ABB RobotStudio station: Demo FlexLoader.rspag

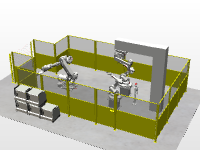
--- station ---
Station Demo FlexLoader (saved by RobotStudio 6.4.7096.126)
Controller Flexloader
  mechanical unit ROB_1: IRB6700_175_305__R1, 6 joints, base frame (0, 0, 0) mm
  mechanical unit ROB_2: IRB1600_6_145__R2, 6 joints, base frame (3100, -700, 540) mm, rotated rx 0 ry 0 rz 180 deg
  mechanical unit ROB_3: IRB1600_6_145__R3, 6 joints, base frame (3100, 700, 540) mm, rotated rx 0 ry 0 rz 180 deg
  mechanical unit ROB_4: IRB1600_6_145__R4, 6 joints, base frame (3100, 0, 2967) mm, rotated rx 180 ry 0 rz 180 deg
Layout (positions relative to the parent item):
  - PKI_500_di_M2001_R2 [mechanism, from Tools\PKI_500_di_M2001.rslib] at (2798.48, -669.1, 1835.93) mm, rotated rx 133.14 ry 80.29 rz -55.34 deg
  - PKI_500_di_M2001_R3 [mechanism, from Tools\PKI_500_di_M2001.rslib] at (2852.02, 663.13, 1854.7) mm, rotated rx -145.04 ry 81.85 rz 49.38 deg
  - PKI_500_di_M2001_R4 [mechanism, from Tools\PKI_500_di_M2001.rslib] at (3569.99, -25.32, 1662.65) mm, rotated rx 170.83 ry -31.84 rz -4.26 deg
  - balk [part] at (-1606.02, -38.05, 675.61) mm, rotated rx -179.44 ry -15.29 rz 176.39 deg
  - FixColumn [part] at (4831, 233, -8) mm, rotated rx 0 ry 0 rz -90 deg
  - RobotStand_2 [part] at (3123, -700, 0) mm, rotated rx 0 ry 0 rz 180 deg
  - RobotStand_3 [part] at (3130, 700, 0) mm, rotated rx 0 ry 0 rz 180 deg
  - IRC5_FlexController_1 [part, from Equipment\IRC5_Control-Module.rslib] at (0, -3200, 100) mm, rotated rx 90 ry 0 rz 0 deg
  - IRC5_DriveModule_1 [part, from Equipment\IRC5_Drive-Module.rslib] at (-750, -3200, 100) mm, rotated rx 90 ry 0 rz 0 deg
  - IRC5_DriveModule_2 [part, from Equipment\IRC5_Drive-Module.rslib] at (-750, -3200, 750) mm, rotated rx 90 ry 0 rz 0 deg
  - IRC5_DriveModule_3 [part, from Equipment\IRC5_Drive-Module.rslib] at (0, -3200, 750) mm, rotated rx 90 ry 0 rz 0 deg
  - IRC5_DriveModule_4 [part, from Equipment\IRC5_Drive-Module.rslib] at (750, -3200, 100) mm, rotated rx 90 ry 0 rz 0 deg
  - IRB1600_6_145__R2 [mechanism, from Robots\IRB1600_6_145_G_02.rslib] at (3100, -700, 540) mm, rotated rx 0 ry 0 rz 180 deg; joint values [-0.0917, -0.6874, 0.2096, -0.087, 0.5953, 0.202] (rad or m)
  - IRB1600_6_145__R3 [mechanism, from Robots\IRB1600_6_145_G_02.rslib] at (3100, 700, 540) mm, rotated rx 0 ry 0 rz 180 deg; joint values [0.1133, -0.7396, 0.1798, 0.2099, 0.6882, -0.2606] (rad or m)
  - IRB1600_6_145__R4 [mechanism, from Robots\IRB1600_6_145_G_02.rslib] at (3100, 0, 2967) mm, rotated rx 180 ry 0 rz 180 deg; joint values [0.0285, -1.3249, -0.0923, 0.2805, -0.7223, 2.9683] (rad or m)
  - IRB6700_175_305__R1 [mechanism, from Robots\IRB6700_175_305__04.rslib] at (0, 0, 0) mm; joint values [0.0254, -0.5043, -3.1116, -0.0184, -0.8299, 0.0976] (rad or m)
  - Fence [graphiccomponentgroup]
    - Segment 1 [part]
    - Segment 2 [part]
    - Segment 3 [part]
    - Segment 4 [part]
    - Segment 5 [part]
    - Segment 6 [part]
    - Segment 7 [part]
    - Segment 8 [part]
    - Segment 9 [part]
    - Segment 10 [part]
    - Segment 11 [part]
    - Segment 12 [part]
    - Segment 13 [part]
    - Segment 14 [part]
    - Segment 15 [part]
    - Segment 16 [part]
    - Segment 17 [part]
  - Floor [part]
  - TSC2013 [mechanism] at (3966.38, 33.42, 0) mm; joint values [1.225] (rad or m)
      links: L1, L2
  - LightGuard [graphiccomponentgroup]
    - GeneratedPart [part] at (-3200, -1000, 200) mm, rotated rx 0 ry 90 rz 90 deg
    - GeneratedPart [part] at (-3200, -1000, 250) mm, rotated rx 0 ry 90 rz 90 deg
    - GeneratedPart [part] at (-3200, -1000, 300) mm, rotated rx 0 ry 90 rz 90 deg
    - GeneratedPart [part] at (-3200, -1000, 350) mm, rotated rx 0 ry 90 rz 90 deg
    - GeneratedPart [part] at (-3200, -1000, 400) mm, rotated rx 0 ry 90 rz 90 deg
    - GeneratedPart [part] at (-3200, -1000, 450) mm, rotated rx 0 ry 90 rz 90 deg
    - GeneratedPart [part] at (-3200, -1000, 500) mm, rotated rx 0 ry 90 rz 90 deg
    - GeneratedPart [part] at (-3200, -1000, 550) mm, rotated rx 0 ry 90 rz 90 deg
    - GeneratedPart [part] at (-3200, -1000, 600) mm, rotated rx 0 ry 90 rz 90 deg
    - GeneratedPart [part] at (-3200, -1000, 650) mm, rotated rx 0 ry 90 rz 90 deg
    - GeneratedPart [part] at (-3200, -1000, 700) mm, rotated rx 0 ry 90 rz 90 deg
    - GeneratedPart [part] at (-3200, -1000, 750) mm, rotated rx 0 ry 90 rz 90 deg
    - GeneratedPart [part] at (-3200, -1000, 800) mm, rotated rx 0 ry 90 rz 90 deg
    - GeneratedPart [part] at (-3200, -1000, 850) mm, rotated rx 0 ry 90 rz 90 deg
    - GeneratedPart [part] at (-3200, -1000, 900) mm, rotated rx 0 ry 90 rz 90 deg
    - GeneratedPart [part] at (-3200, -1000, 950) mm, rotated rx 0 ry 90 rz 90 deg
    - GeneratedPart [part] at (-3200, -1000, 1000) mm, rotated rx 0 ry 90 rz 90 deg
    - GeneratedPart [part] at (-3200, -1000, 1050) mm, rotated rx 0 ry 90 rz 90 deg
    - GeneratedPart [part] at (-3200, -1000, 1100) mm, rotated rx 0 ry 90 rz 90 deg
    - GeneratedPart [part] at (-3200, -1000, 1150) mm, rotated rx 0 ry 90 rz 90 deg
    - GeneratedPart [part] at (-3200, -1000, 1200) mm, rotated rx 0 ry 90 rz 90 deg
    - GeneratedPart [part] at (-3200, -1000, 1250) mm, rotated rx 0 ry 90 rz 90 deg
    - GeneratedPart [part] at (-3200, -1000, 1300) mm, rotated rx 0 ry 90 rz 90 deg
    - GeneratedPart [part] at (-3200, -1000, 1350) mm, rotated rx 0 ry 90 rz 90 deg
    - GeneratedPart [part] at (-3200, -1000, 1400) mm, rotated rx 0 ry 90 rz 90 deg
    - GeneratedPart [part] at (-3200, -1000, 1450) mm, rotated rx 0 ry 90 rz 90 deg
    - GeneratedPart [part] at (-3200, -1000, 1500) mm, rotated rx 0 ry 90 rz 90 deg
    - GeneratedPart [part] at (-3200, -1000, 1550) mm, rotated rx 0 ry 90 rz 90 deg
    - GeneratedPart [part] at (-3200, -1000, 1600) mm, rotated rx 0 ry 90 rz 90 deg
    - GeneratedPart [part] at (-3200, -1000, 1650) mm, rotated rx 0 ry 90 rz 90 deg
    - GeneratedPart [part] at (-3200, -1000, 1700) mm, rotated rx 0 ry 90 rz 90 deg
    - GeneratedPart [part] at (-3200, -1000, 1750) mm, rotated rx 0 ry 90 rz 90 deg
    - light_guard1 [part] at (-3200, -1000, 0) mm, rotated rx 0 ry 0 rz 90 deg
    - light_guard2 [part] at (-3200, 1000, 0) mm, rotated rx 0 ry 0 rz 90 deg
  - R1 [frame] at (3100, -700, 540) mm, rotated rx 0 ry 0 rz 180 deg
  - R2 [frame] at (3100, 700, 540) mm, rotated rx 0 ry 0 rz 180 deg
  - R3 [frame] at (3100, 0, 2967) mm, rotated rx 180 ry 0 rz 180 deg
  - R4 [frame]
  - Frame_5 [frame] at (1912, 0, 2055) mm, rotated rx 0 ry 90 rz 0 deg
  - Frame_1 [frame] at (-1606.02, -38.05, 675.61) mm, rotated rx -179.44 ry -15.29 rz 176.39 deg
  - Frame_2 [frame]
Attachment: PKI_500_di_M2001_R2 is attached to IRB1600_6_145__R2 / Link6
Attachment: PKI_500_di_M2001_R3 is attached to IRB1600_6_145__R3 / Link6
Attachment: PKI_500_di_M2001_R4 is attached to IRB1600_6_145__R4 / Link6
Attachment: balk is attached to IRB6700_175_305__R1 / Link6
Targets, tools, work objects and paths stored in the station and not in the controller backup, written as RAPID:
! task T_ROB1
MODULE Module1
  CONST robtarget Target_10:=[[1912,0,2055],[0.707106781,0,0.707106781,0],[0,0,0,0],[9E+09,9E+09,9E+09,9E+09,9E+09,9E+09]];
  VAR syncident ident1;
  VAR syncident ident2;
  VAR syncident ident3;
  VAR syncident ident4;
  VAR syncident ident5;
  VAR syncident ident6;
  VAR syncident ident7;
  VAR syncident ident8;
  VAR syncident ident9;
ENDMODULE

! task T_ROB2
MODULE Module1
  VAR syncident ident1;
  VAR syncident ident2;
  VAR syncident ident3;
  VAR syncident ident4;
  VAR syncident ident5;
  VAR syncident ident6;
  VAR syncident ident7;
  VAR syncident ident8;
  VAR syncident ident9;
  VAR syncident identUnder1;
  VAR syncident identUnder2;
  VAR syncident identEdge1;
  VAR syncident identEdge2;
  VAR syncident identCurve1;
  VAR syncident identCurve2;
  VAR syncident identBack1;
  VAR syncident identBack2;
  VAR syncident identTop1;
  VAR syncident identTop2;
  VAR syncident identRing1;
  VAR syncident identRing2;
ENDMODULE

! task T_ROB3
MODULE Module1
  VAR syncident ident1;
  VAR syncident ident2;
  VAR syncident ident3;
  VAR syncident ident4;
  VAR syncident ident5;
  VAR syncident ident6;
  VAR syncident ident7;
  VAR syncident ident8;
  VAR syncident ident9;
  VAR syncident identUnder1;
  VAR syncident identUnder2;
  VAR syncident identEdge1;
  VAR syncident identEdge2;
  VAR syncident identCurve1;
  VAR syncident identCurve2;
  VAR syncident identBack1;
  VAR syncident identBack2;
  VAR syncident identTop1;
  VAR syncident identTop2;
  VAR syncident identRing1;
  VAR syncident identRing2;
ENDMODULE

! task T_ROB4
MODULE module1
  VAR syncident ident1;
  VAR syncident ident2;
  VAR syncident ident3;
  VAR syncident ident4;
  VAR syncident ident5;
  VAR syncident ident6;
  VAR syncident ident7;
  VAR syncident ident8;
  VAR syncident ident9;
  VAR syncident identEdge1;
  VAR syncident identEdge2;
  VAR syncident identTop1;
  VAR syncident identTop2;
ENDMODULE


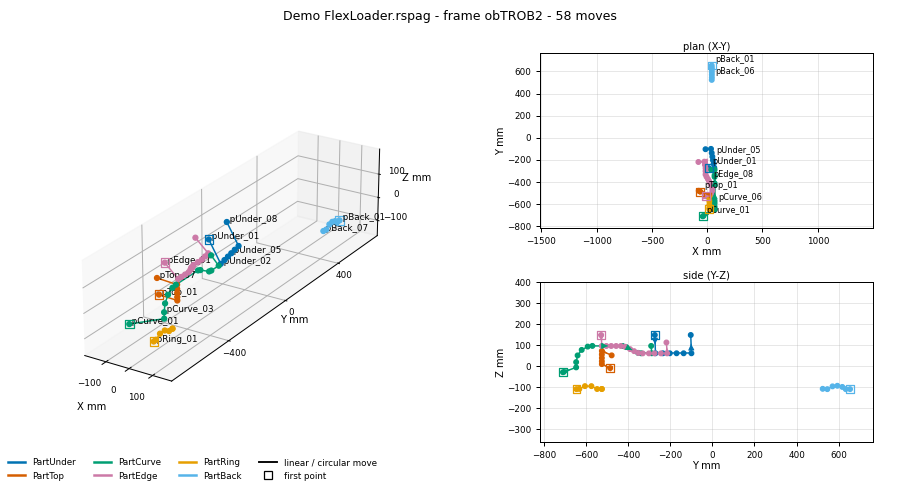
[picture p0: tool path of Demo FlexLoader.rspag in frame obTROB2, 58 of 166 moves have a stored position in this frame; points joined in program order, loops and branches not executed]
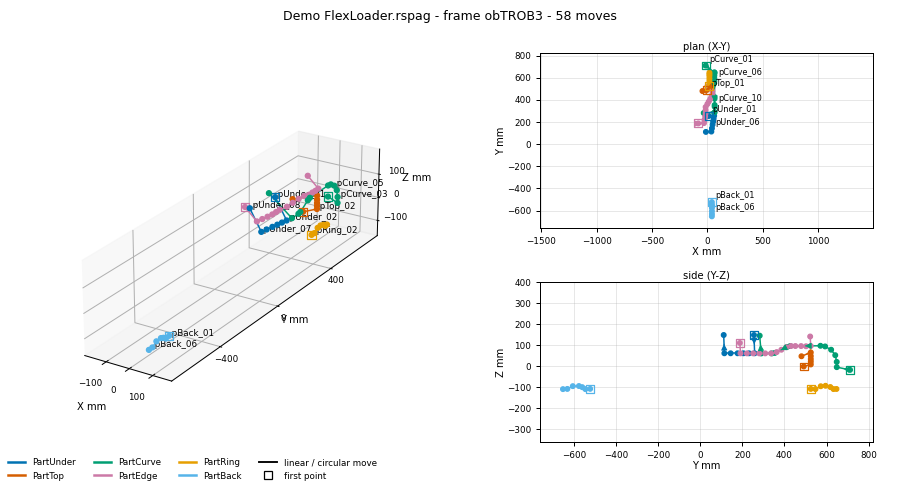
[picture p1: tool path of Demo FlexLoader.rspag in frame obTROB3, 58 of 166 moves have a stored position in this frame; points joined in program order, loops and branches not executed]
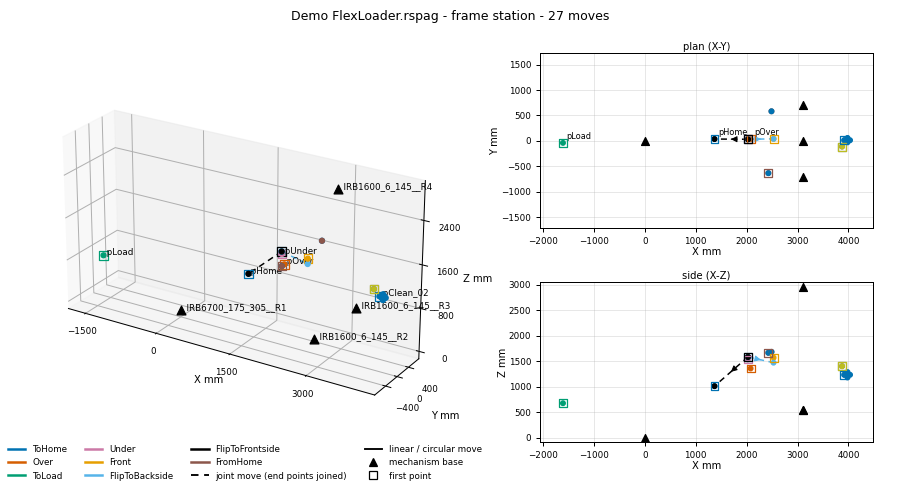
[picture p2: tool path of Demo FlexLoader.rspag in frame station, 27 of 166 moves have a stored position in this frame; points joined in program order, loops and branches not executed]
--- Backups/Flexloader/RAPID/TASK1/PROGMOD/Module1.mod ---
%%%
   VERSION: 1
   LANGUAGE: ENGLISH
%%%

MODULE Module1
	VAR syncident ident1;
	PERS tasks task1{4}:=[["T_ROB1"],["T_ROB2"],["T_ROB3"],["T_ROB4"]];
	VAR syncident ident2;
	VAR syncident ident3;
	VAR syncident ident4;
	VAR syncident ident5;
	VAR syncident ident6;
	PERS tasks task4{3}:=[["T_ROB1"],["T_ROB2"],["T_ROB3"]];
	VAR syncident ident7;
	VAR syncident ident8;
	VAR syncident ident9;
	CONST robtarget pHome:=[[1369.512905465,37.466644332,1010.783503591],[0.745592277,0.014819779,0.664663533,0.045770282],[0,-1,0,1],[9E+09,9E+09,9E+09,9E+09,9E+09,9E+09]];
	CONST robtarget pOver:=[[2078.60907176,35.539251508,1357.923045634],[0.636059947,-0.027312722,0.771147463,-0.00365378],[0,-1,0,1],[9E+09,9E+09,9E+09,9E+09,9E+09,9E+09]];
	CONST robtarget pLoad:=[[-1606.023702637,-38.0457751,675.609388963],[0.133106755,-0.030537275,-0.99063094,0.000638774],[0,-1,0,7],[9E+09,9E+09,9E+09,9E+09,9E+09,9E+09]];
	CONST robtarget pUnder:=[[2026.430172321,41.745619209,1534.299517082],[0.919452647,-0.027776408,0.392048067,0.011559176],[0,-1,0,1],[9E+09,9E+09,9E+09,9E+09,9E+09,9E+09]];
	CONST robtarget pFront:=[[2530.563907646,41.394092958,1569.72454293],[0.492426348,0.001222862,0.870261855,0.012613516],[0,0,0,0],[9E+09,9E+09,9E+09,9E+09,9E+09,9E+09]];
	CONST robtarget pFlip_01:=[[2026.542021706,32.724801885,1584.151071251],[0.522506749,0.002471091,0.852548409,0.011908016],[0,0,0,0],[9E+09,9E+09,9E+09,9E+09,9E+09,9E+09]];
	CONST robtarget pFlip_02:=[[2026.542021706,32.724801885,1584.151071251],[0.011908016,-0.852548409,0.002471091,-0.522506749],[0,0,2,0],[9E+09,9E+09,9E+09,9E+09,9E+09,9E+09]];
	CONST robtarget pFlip_03:=[[2528.820790114,41.134978002,1471.579982878],[0.012222966,-0.870264365,0.001710031,-0.49243031],[0,0,2,0],[9E+09,9E+09,9E+09,9E+09,9E+09,9E+09]];

PROC main()
	ToHome;
	Over;
	WaitSyncTask ident1,task1;
	WaitSyncTask ident2,task1;
	Under;
	WaitSyncTask ident3,task1;
	WaitSyncTask ident4,task1;
	WaitSyncTask ident5,task1;
	Front;
	WaitSyncTask ident6,task1;
	WaitSyncTask ident7,task1;
	FlipToBackside;
	WaitSyncTask ident8,task1;
	WaitSyncTask ident9,task1;
	FlipToFrontside;
	ToLoad;
ENDPROC

PROC ToHome()
	MoveJ pHome,vmax,fine,tool0\WObj:=wobj0;
ENDPROC

PROC Over()
	MoveJ pOver,vmax,fine,tool0\WObj:=wobj0;
ENDPROC

PROC ToLoad()
	MoveJ pLoad,vmax,fine,tool0\WObj:=wobj0;
ENDPROC

PROC Under()
	MoveJ pUnder,vmax,fine,tool0\WObj:=wobj0;
ENDPROC

PROC Front()
	MoveJ pFront,v1000,fine,tool0\WObj:=wobj0;
ENDPROC

PROC FlipToBackside()
	MoveJ pFlip_01,v1000,z100,tool0\WObj:=wobj0;
	MoveJ pFlip_02,v1000,z100,tool0\WObj:=wobj0;
	MoveJ pFlip_03,v1000,fine,tool0\WObj:=wobj0;
ENDPROC

PROC FlipToFrontside()
	MoveJ pFlip_02,v1000,z100,tool0\WObj:=wobj0;
	MoveJ pFlip_01,v1000,z100,tool0\WObj:=wobj0;
	MoveJ pHome,v1000,z100,tool0\WObj:=wobj0;
ENDPROC
ENDMODULE

--- Backups/Flexloader/RAPID/TASK1/SYSMOD/LINKEDM.sys ---
%%%
  VERSION:1
  LANGUAGE:ENGLISH
%%%

MODULE LINKEDM (SYSMODULE)

! FOLLOWER
!     Name of electronically linked follower axis used by operator at teach pendent.
      PERS string l_f_axis_name{5}       :=  ["",  "", "", "", ""];

!     Name of the mechanical unit for follower axis.
      PERS string l_f_mecunt_n{5}  :=  ["", "", "", "", ""];

!     Linked follower axis number in the mechanical unit (first axis in mech. unit is number 1).
      PERS num l_f_axis_no{5}      :=  [0,          0,   0,  0,  0];

! MASTER
!     Name of the mechanical unit for linked master axis.
      PERS string l_m_mecunt_n{5} :=  ["", "", "", "", ""];

!     Linked master axis number in the mechanical unit (first axis in mech. unit is number 1).
!     See axis number table in documentation for different master mechanical units.
      PERS num l_m_axis_no{5}     :=  [0,  0,  0,  0,  0];

! POSITION OFFSET
!     The increase of the allowed offset position between the master and follower
!     positions, used when starting AUTO mode. As soon as the offset is decreased
!     the old configurated parameter is used.
!     Example: 3 => the configurated value of allowed offset is increased 3 times.
      PERS num offset_ratio{5}       :=  [10,  10,   10,  10,  10];

! SPEED RATIO
!     Speed_ratio used in AUTO and JOG modes [ very_slow   slow    normal    fast]
!     Value 1 = max allowed manual speed.
      CONST num speed_ratio {20}      := [0.01, 0.01, 0.01, 0.01, 0.01,
                                          0.05, 0.05, 0.05, 0.05, 0.05,
                                          0.20, 0.20, 0.20, 0.20, 0.20,
                                          1.00, 1.00, 1.00, 1.00, 1.00];

! STEP SIZE
!     Displacement position used in JOG mode for each activation of positive or
!     negative movement.                  [very_short    short   normal   long]
!     Unit degees or meter.
      CONST num displacement {20}     := [0.001, 0.001, 0.001, 0.001, 0.001,
                                          0.005, 0.005, 0.005, 0.005, 0.005,
                                          0.020, 0.020, 0.020, 0.020, 0.020,
                                          0.100, 0.100, 0.100, 0.100, 0.100];


!-------------------------------------------------------------
 PROC Linked_m ()
      Linked_m_exe ;
 ENDPROC
ENDMODULE

--- Backups/Flexloader/RAPID/TASK2/PROGMOD/Module1.mod ---
%%%
   VERSION: 1
   LANGUAGE: ENGLISH
%%%

MODULE Module1
	VAR syncident ident1;
	PERS tasks task1{4}:=[["T_ROB1"],["T_ROB2"],["T_ROB3"],["T_ROB4"]];
	VAR syncident ident2;
	VAR syncident ident3;
	VAR syncident ident4;
	VAR syncident ident5;
	VAR syncident ident6;
	PERS tasks task4{3}:=[["T_ROB1"],["T_ROB2"],["T_ROB3"]];
	VAR syncident ident7;
	VAR syncident ident8;
	VAR syncident ident9;
	CONST robtarget pUnder_01:=[[14.958979691,-273.413172673,148.825312372],[0.017229453,-0.96649232,0.004340926,-0.256079867],[-1,0,-1,0],[9E+09,9E+09,9E+09,9E+09,9E+09,9E+09]];
	PERS tooldata PKI_500:=[TRUE,[[126.925343398,0,389.787472308],[0.898794046,0,0.438371147,0]],[1,[0,0,0.1],[1,0,0,0],0,0,0]];
	PERS wobjdata obTROB2:=[FALSE,FALSE,"ROB_1",[[0,0,0],[1,0,0,0]],[[0,0,0],[1,0,0,0]]];
	VAR syncident identUnder1;
	PERS tasks task2{2}:=[["T_ROB2"],["T_ROB3"]];
	CONST robtarget pUnder_02:=[[64.473645199,-270.305046432,62],[0.017229379,-0.966492374,0.004340901,-0.256079667],[-1,0,-1,0],[9E+09,9E+09,9E+09,9E+09,9E+09,9E+09]];
	CONST robtarget pUnder_03:=[[58.303525946,-235.207684857,62],[0.017229379,-0.966492374,0.004340901,-0.256079667],[-1,0,-1,0],[9E+09,9E+09,9E+09,9E+09,9E+09,9E+09]];
	CONST robtarget pUnder_04:=[[52.509460014,-202.249419606,62],[0.017229379,-0.966492374,0.004340901,-0.256079667],[-1,0,-1,0],[9E+09,9E+09,9E+09,9E+09,9E+09,9E+09]];
	CONST robtarget pUnder_05:=[[46.857542536,-170.099734462,62],[0.017229379,-0.966492374,0.004340901,-0.256079667],[-1,0,-1,0],[9E+09,9E+09,9E+09,9E+09,9E+09,9E+09]];
	CONST robtarget pUnder_06:=[[40.944873567,-136.466822007,62],[0.017229379,-0.966492374,0.004340901,-0.256079667],[-1,0,-1,0],[9E+09,9E+09,9E+09,9E+09,9E+09,9E+09]];
	CONST robtarget pUnder_07:=[[34.463035646,-99.596317592,62],[0.017229379,-0.966492374,0.004340901,-0.256079667],[-1,0,-1,0],[9E+09,9E+09,9E+09,9E+09,9E+09,9E+09]];
	CONST robtarget pUnder_08:=[[-15.051684524,-102.704337479,148.825314878],[0.017229359,-0.966492315,0.004340943,-0.256079891],[-1,0,-1,0],[9E+09,9E+09,9E+09,9E+09,9E+09,9E+09]];
	VAR syncident identUnder2;
	CONST robtarget pHome:=[[2427.29581164,-632.400445714,1665.867539911],[0.038314456,0.956854288,-0.091070705,-0.27325446],[-1,-1,0,0],[9E+09,9E+09,9E+09,9E+09,9E+09,9E+09]];
	CONST robtarget pTop_01:=[[-63.846269958,-485.429084696,-8.338300316],[0.19188065,0.607043211,-0.260314366,0.725890341],[-1,0,-1,0],[9E+09,9E+09,9E+09,9E+09,9E+09,9E+09]];
	CONST robtarget pTop_02:=[[42,-525,10.577955055],[0.19188065,0.607043211,-0.260314366,0.725890341],[-1,0,-1,0],[9E+09,9E+09,9E+09,9E+09,9E+09,9E+09]];
	VAR syncident identTop1;
	PERS tasks task3{3}:=[["T_ROB2"],["T_ROB3"],["T_ROB4"]];
	CONST robtarget pTop_03:=[[42,-525,23.953188676],[0.19188065,0.607043211,-0.260314366,0.725890341],[-1,0,-1,0],[9E+09,9E+09,9E+09,9E+09,9E+09,9E+09]];
	CONST robtarget pTop_04:=[[42,-525,39.706941228],[0.19188065,0.607043211,-0.260314366,0.725890341],[-1,0,-1,0],[9E+09,9E+09,9E+09,9E+09,9E+09,9E+09]];
	CONST robtarget pTop_05:=[[42,-525,56.305032418],[0.19188065,0.607043211,-0.260314366,0.725890341],[-1,0,-1,0],[9E+09,9E+09,9E+09,9E+09,9E+09,9E+09]];
	CONST robtarget pTop_06:=[[42,-525,73.146723771],[0.19188065,0.607043211,-0.260314366,0.725890341],[-1,0,-1,0],[9E+09,9E+09,9E+09,9E+09,9E+09,9E+09]];
	VAR syncident identTop2;
	CONST robtarget pTop_07:=[[-76.280174357,-478.382735403,52.099937261],[0.19188065,0.607043211,-0.260314366,0.725890341],[-1,0,-1,0],[9E+09,9E+09,9E+09,9E+09,9E+09,9E+09]];
	CONST robtarget pCurve_01:=[[-40.080509268,-709.629888972,-28.057934223],[0.328524284,-0.791658328,0.18277424,-0.481604053],[0,0,-1,1],[9E+09,9E+09,9E+09,9E+09,9E+09,9E+09]];
	VAR syncident identCurve1;
	CONST robtarget pCurve_02:=[[67.000045259,-646.999937599,-4.999944365],[0.328524284,-0.791658328,0.18277424,-0.481604053],[0,0,-1,1],[9E+09,9E+09,9E+09,9E+09,9E+09,9E+09]];
	CONST robtarget pCurve_03:=[[66.999941382,-646.999939722,20.000055537],[0.328524284,-0.791658328,0.18277424,-0.481604053],[0,0,-1,1],[9E+09,9E+09,9E+09,9E+09,9E+09,9E+09]];
	CONST robtarget pCurve_04:=[[66.999982099,-640.112495856,51.831340748],[0.328524284,-0.791658328,0.18277424,-0.481604053],[0,0,-1,1],[9E+09,9E+09,9E+09,9E+09,9E+09,9E+09]];
	CONST robtarget pCurve_05:=[[66.999899596,-620.682247644,77.968115009],[0.328524284,-0.791658328,0.18277424,-0.481604053],[0,0,-1,1],[9E+09,9E+09,9E+09,9E+09,9E+09,9E+09]];
	CONST robtarget pCurve_06:=[[66.999897769,-592.185311674,93.734869346],[0.328524284,-0.791658328,0.18277424,-0.481604053],[0,0,-1,1],[9E+09,9E+09,9E+09,9E+09,9E+09,9E+09]];
	CONST robtarget pCurve_07:=[[66.999906472,-569.999933514,97.000138844],[0.328524284,-0.791658328,0.18277424,-0.481604053],[0,0,-1,1],[9E+09,9E+09,9E+09,9E+09,9E+09,9E+09]];
	CONST robtarget pCurve_08:=[[66.999884239,-426.268505537,96.673140898],[0.328524284,-0.791658328,0.18277424,-0.481604053],[-1,0,-1,1],[9E+09,9E+09,9E+09,9E+09,9E+09,9E+09]];
	CONST robtarget pCurve_09:=[[66.999892662,-410.784253533,92.03826085],[0.27883297,-0.805661501,0.163375852,-0.496457502],[-1,0,-1,1],[9E+09,9E+09,9E+09,9E+09,9E+09,9E+09]];
	CONST robtarget pCurve_10:=[[66.999819776,-352.977721713,64.103032003],[0.223102529,-0.818032773,0.141414351,-0.510930157],[-1,0,-1,1],[9E+09,9E+09,9E+09,9E+09,9E+09,9E+09]];
	CONST robtarget pCurve_11:=[[66.999894322,-338.196479113,62.000174956],[0.280217315,-0.805310116,0.163918658,-0.496069095],[-1,0,-1,1],[9E+09,9E+09,9E+09,9E+09,9E+09,9E+09]];
	CONST robtarget pCurve_12:=[[66.999906799,-288.222073771,62.000218277],[0.328524284,-0.791658328,0.18277424,-0.481604053],[-1,0,-1,1],[9E+09,9E+09,9E+09,9E+09,9E+09,9E+09]];
	VAR syncident identCurve2;
	CONST robtarget pCurve_13:=[[35.872289812,-290.698064532,96.909414765],[0.328524284,-0.791658328,0.18277424,-0.481604053],[-1,0,-1,1],[9E+09,9E+09,9E+09,9E+09,9E+09,9E+09]];
	CONST robtarget pEdge_01:=[[-7.327915766,-528.236933692,148.557107932],[0.025535838,-0.989726688,0.004582217,-0.140598745],[-1,0,-1,0],[9E+09,9E+09,9E+09,9E+09,9E+09,9E+09]];
	VAR syncident identEdge1;
	CONST robtarget pEdge_02:=[[46.916281985,-525.078505399,96.60776602],[0.025535862,-0.989726678,0.004582193,-0.140598813],[-1,0,-1,0],[9E+09,9E+09,9E+09,9E+09,9E+09,9E+09]];
	CONST robtarget pEdge_03:=[[47.117343896,-503.71339074,96.607981897],[0.025535799,-0.989726681,0.004582226,-0.1405988],[-1,0,-1,0],[9E+09,9E+09,9E+09,9E+09,9E+09,9E+09]];
	CONST robtarget pEdge_04:=[[47.115988899,-480.469842231,96.608479881],[0.025535853,-0.989726681,0.004582209,-0.140598796],[-1,0,-1,0],[9E+09,9E+09,9E+09,9E+09,9E+09,9E+09]];
	CONST robtarget pEdge_05:=[[47.114567358,-457.1247098,96.60882774],[0.025535818,-0.989726679,0.00458223,-0.140598812],[-1,0,-1,0],[9E+09,9E+09,9E+09,9E+09,9E+09,9E+09]];
	CONST robtarget pEdge_06:=[[40.19468128,-434.661991273,96.609447443],[0.025535863,-0.98972668,0.004582221,-0.140598799],[-1,0,-1,0],[9E+09,9E+09,9E+09,9E+09,9E+09,9E+09]];
	CONST robtarget pEdge_07:=[[29.704287715,-414.145572252,92.882126466],[0.025535851,-0.989726679,0.004582203,-0.140598807],[-1,0,-1,0],[9E+09,9E+09,9E+09,9E+09,9E+09,9E+09]];
	CONST robtarget pEdge_08:=[[16.852998769,-390.944921934,81.750547877],[0.025535844,-0.989726681,0.004582204,-0.140598795],[-1,0,-1,0],[9E+09,9E+09,9E+09,9E+09,9E+09,9E+09]];
	CONST robtarget pEdge_09:=[[6.006560889,-371.669455014,72.113178486],[0.025535805,-0.989726684,0.004582248,-0.140598781],[-1,0,-1,0],[9E+09,9E+09,9E+09,9E+09,9E+09,9E+09]];
	CONST robtarget pEdge_10:=[[-5.937544655,-351.427181731,63.426760138],[0.025535812,-0.989726684,0.004582232,-0.140598778],[-1,0,-1,0],[9E+09,9E+09,9E+09,9E+09,9E+09,9E+09]];
	CONST robtarget pEdge_11:=[[-14.847685459,-330.777409413,61.612404686],[0.025535835,-0.989726682,0.004582227,-0.140598791],[-1,0,-1,0],[9E+09,9E+09,9E+09,9E+09,9E+09,9E+09]];
	CONST robtarget pEdge_12:=[[-14.849542018,-301.436386394,61.612910705],[0.025535821,-0.989726683,0.004582226,-0.140598786],[-1,0,-1,0],[9E+09,9E+09,9E+09,9E+09,9E+09,9E+09]];
	CONST robtarget pEdge_13:=[[-14.851261771,-274.659068574,61.613232611],[0.025535843,-0.989726679,0.004582226,-0.14059881],[-1,0,-1,0],[9E+09,9E+09,9E+09,9E+09,9E+09,9E+09]];
	CONST robtarget pEdge_14:=[[-20.172939671,-244.399635183,61.614002493],[0.025535864,-0.989726679,0.004582214,-0.140598803],[-1,0,-1,0],[9E+09,9E+09,9E+09,9E+09,9E+09,9E+09]];
	CONST robtarget pEdge_15:=[[-25.338508764,-215.027453723,61.614581797],[0.025535833,-0.989726679,0.004582212,-0.140598809],[-1,0,-1,0],[9E+09,9E+09,9E+09,9E+09,9E+09,9E+09]];
	VAR syncident identEdge2;
	CONST robtarget pEdge_16:=[[-79.321708087,-218.170721913,113.314114025],[0.025535838,-0.989726688,0.004582217,-0.140598745],[-1,0,-1,0],[9E+09,9E+09,9E+09,9E+09,9E+09,9E+09]];
	VAR syncident identRing1;
	CONST robtarget pRing_01:=[[19.488526003,-645.518538398,-108.232346635],[0.062664951,-0.707787609,0.090592708,-0.697784183],[-1,0,-1,0],[9E+09,9E+09,9E+09,9E+09,9E+09,9E+09]];
	CONST robtarget pRing_02:=[[19.487710187,-631.852499886,-107.23742612],[0.062664947,-0.707787603,0.090592717,-0.697784188],[-1,0,-1,0],[9E+09,9E+09,9E+09,9E+09,9E+09,9E+09]];
	CONST robtarget pRing_03:=[[19.486358866,-605.247177595,-94.028087652],[0.06266495,-0.707787588,0.090592715,-0.697784203],[-1,0,-1,0],[9E+09,9E+09,9E+09,9E+09,9E+09,9E+09]];
	CONST robtarget pRing_04:=[[19.484320741,-574.613939637,-94.038595956],[0.062664937,-0.707787594,0.090592731,-0.697784196],[-1,0,-1,0],[9E+09,9E+09,9E+09,9E+09,9E+09,9E+09]];
	CONST robtarget pRing_05:=[[19.482238078,-547.479258887,-107.713968108],[0.062664928,-0.707787592,0.090592731,-0.697784199],[-1,0,-1,0],[9E+09,9E+09,9E+09,9E+09,9E+09,9E+09]];
	CONST robtarget pRing_06:=[[19.480879155,-524.953352106,-107.518283993],[0.062664949,-0.707787587,0.090592712,-0.697784204],[-1,0,-1,0],[9E+09,9E+09,9E+09,9E+09,9E+09,9E+09]];
	CONST robtarget pRing_07:=[[19.480879155,-524.953352106,-107.518283993],[0.062664949,-0.707787587,0.090592712,-0.697784204],[-1,0,-1,0],[9E+09,9E+09,9E+09,9E+09,9E+09,9E+09]];
	VAR syncident identRing2;
	VAR syncident identBack1;
	CONST robtarget pBack_01:=[[41.260544477,653.762434597,-108.211687392],[0.697844958,-0.090352613,-0.707808862,0.062092147],[-1,0,0,0],[9E+09,9E+09,9E+09,9E+09,9E+09,9E+09]];
	CONST robtarget pBack_02:=[[41.952428022,633.411421546,-108.159146012],[0.697844972,-0.090352612,-0.707808848,0.062092149],[-1,0,-1,0],[9E+09,9E+09,9E+09,9E+09,9E+09,9E+09]];
	CONST robtarget pBack_03:=[[41.943862758,617.021990928,-97.800743575],[0.697844972,-0.090352626,-0.707808847,0.062092145],[-1,0,-1,0],[9E+09,9E+09,9E+09,9E+09,9E+09,9E+09]];
	CONST robtarget pBack_04:=[[41.953948167,593.539459054,-92.317425881],[0.697844979,-0.09035262,-0.707808841,0.06209215],[-1,0,-1,0],[9E+09,9E+09,9E+09,9E+09,9E+09,9E+09]];
	CONST robtarget pBack_05:=[[41.953651293,570.640431166,-95.107229688],[0.697844983,-0.090352631,-0.707808836,0.062092147],[-1,0,-1,0],[9E+09,9E+09,9E+09,9E+09,9E+09,9E+09]];
	CONST robtarget pBack_06:=[[41.951803799,545.854793959,-108.331667407],[0.697844973,-0.0903526,-0.707808849,0.062092151],[-1,0,-1,0],[9E+09,9E+09,9E+09,9E+09,9E+09,9E+09]];
	CONST robtarget pBack_07:=[[41.304365327,524.004978144,-106.769191783],[0.697844979,-0.090352631,-0.707808839,0.062092144],[-1,0,-1,0],[9E+09,9E+09,9E+09,9E+09,9E+09,9E+09]];
	VAR syncident identBack2;

PROC main()
	WaitSyncTask ident1,task1;
	FromHome;
	PartTop;
	PartCurve;
	ToHome;
	WaitSyncTask ident2,task1;
	WaitSyncTask ident3,task1;
	FromHome;
	PartUnder;
	WaitSyncTask ident4,task1;
	PartEdge;
	ToHome;
	WaitSyncTask ident5,task1;
	WaitSyncTask ident6,task1;
	FromHome;
	PartRing;
	ToHome;
	WaitSyncTask ident7,task1;
	WaitSyncTask ident8,task1;
	FromHome;
	PartBack;
	ToHome;
	WaitSyncTask ident9,task1;
ENDPROC

PROC PartUnder()
	MoveJ pUnder_01,vmax,fine,PKI_500\WObj:=obTROB2;
	SyncMoveOn identUnder1,task2;
	MoveL pUnder_02\ID:=10,v100,z1,PKI_500\WObj:=obTROB2;
	MoveL pUnder_03\ID:=20,v100,z1,PKI_500\WObj:=obTROB2;
	MoveL pUnder_04\ID:=30,v100,z1,PKI_500\WObj:=obTROB2;
	MoveL pUnder_05\ID:=40,v100,z1,PKI_500\WObj:=obTROB2;
	MoveL pUnder_06\ID:=50,v100,z1,PKI_500\WObj:=obTROB2;
	MoveL pUnder_07\ID:=60,v100,z1,PKI_500\WObj:=obTROB2;
	MoveL pUnder_08\ID:=70,v100,fine,PKI_500\WObj:=obTROB2;
	SyncMoveOff identUnder2;
ENDPROC

PROC FromHome()
	MoveJ pHome,vmax,fine,PKI_500\WObj:=wobj0;
ENDPROC

PROC ToHome()
	MoveJ pHome,vmax,fine,PKI_500\WObj:=wobj0;
ENDPROC

PROC PartTop()
	MoveJ pTop_01,vmax,z100,PKI_500\WObj:=obTROB2;
	MoveL pTop_02,v500,fine,PKI_500\WObj:=obTROB2;
	SyncMoveOn identTop1,task3;
	MoveL pTop_03\ID:=10,v100,z1,PKI_500\WObj:=obTROB2;
	MoveL pTop_04\ID:=20,v100,z1,PKI_500\WObj:=obTROB2;
	MoveL pTop_05\ID:=30,v100,z1,PKI_500\WObj:=obTROB2;
	MoveL pTop_06\ID:=40,v100,fine,PKI_500\WObj:=obTROB2;
	SyncMoveOff identTop2;
	MoveL pTop_07,v500,z100,PKI_500\WObj:=obTROB2;
ENDPROC

PROC PartCurve()
	MoveJ pCurve_01,v1000,z100,PKI_500\WObj:=obTROB2;
	SyncMoveOn identCurve1,task2;
	MoveL pCurve_02\ID:=20,v100,z1,PKI_500\WObj:=obTROB2;
	MoveL pCurve_03\ID:=30,v100,z1,PKI_500\WObj:=obTROB2;
	MoveL pCurve_04\ID:=40,v100,z1,PKI_500\WObj:=obTROB2;
	MoveL pCurve_05\ID:=50,v100,z1,PKI_500\WObj:=obTROB2;
	MoveL pCurve_06\ID:=60,v100,z1,PKI_500\WObj:=obTROB2;
	MoveL pCurve_07\ID:=70,v100,z1,PKI_500\WObj:=obTROB2;
	MoveL pCurve_08\ID:=80,v100,z1,PKI_500\WObj:=obTROB2;
	MoveL pCurve_09\ID:=90,v100,z1,PKI_500\WObj:=obTROB2;
	MoveL pCurve_10\ID:=100,v100,z1,PKI_500\WObj:=obTROB2;
	MoveL pCurve_11\ID:=110,v100,z1,PKI_500\WObj:=obTROB2;
	MoveL pCurve_12\ID:=120,v100,fine,PKI_500\WObj:=obTROB2;
	SyncMoveOff identCurve2;
	MoveL pCurve_13,v500,z100,PKI_500\WObj:=obTROB2;
ENDPROC

PROC PartEdge()
	MoveJ pEdge_01,v1000,fine,PKI_500\WObj:=obTROB2;
	SyncMoveOn identEdge1,task3;
	MoveL pEdge_02\ID:=10,v100,z1,PKI_500\WObj:=obTROB2;
	MoveL pEdge_03\ID:=20,v100,z1,PKI_500\WObj:=obTROB2;
	MoveL pEdge_04\ID:=30,v100,z1,PKI_500\WObj:=obTROB2;
	MoveL pEdge_05\ID:=40,v100,z1,PKI_500\WObj:=obTROB2;
	MoveL pEdge_06\ID:=50,v100,z1,PKI_500\WObj:=obTROB2;
	MoveL pEdge_07\ID:=60,v100,z1,PKI_500\WObj:=obTROB2;
	MoveL pEdge_08\ID:=70,v100,z1,PKI_500\WObj:=obTROB2;
	MoveL pEdge_09\ID:=80,v100,z1,PKI_500\WObj:=obTROB2;
	MoveL pEdge_10\ID:=90,v100,z1,PKI_500\WObj:=obTROB2;
	MoveL pEdge_11\ID:=100,v100,z1,PKI_500\WObj:=obTROB2;
	MoveL pEdge_12\ID:=110,v100,z1,PKI_500\WObj:=obTROB2;
	MoveL pEdge_13\ID:=120,v100,z1,PKI_500\WObj:=obTROB2;
	MoveL pEdge_14\ID:=130,v100,z1,PKI_500\WObj:=obTROB2;
	MoveL pEdge_15\ID:=140,v100,fine,PKI_500\WObj:=obTROB2;
	SyncMoveOff identEdge2;
	MoveL pEdge_16,v1000,z100,PKI_500\WObj:=obTROB2;
ENDPROC

PROC PartRing()
	SyncMoveOn identRing1,task2;
	MoveL pRing_01\ID:=10,v100,z1,PKI_500\WObj:=obTROB2;
	MoveL pRing_02\ID:=20,v100,z1,PKI_500\WObj:=obTROB2;
	MoveL pRing_03\ID:=30,v100,z1,PKI_500\WObj:=obTROB2;
	MoveL pRing_04\ID:=40,v100,z1,PKI_500\WObj:=obTROB2;
	MoveL pRing_05\ID:=50,v100,z1,PKI_500\WObj:=obTROB2;
	MoveL pRing_06\ID:=60,v100,z1,PKI_500\WObj:=obTROB2;
	MoveL pRing_07\ID:=70,v100,fine,PKI_500\WObj:=obTROB2;
	SyncMoveOff identRing2;
ENDPROC

PROC PartBack()
	SyncMoveOn identBack1,task2;
	MoveL pBack_01\ID:=10,v100,z1,PKI_500\WObj:=obTROB2;
	MoveL pBack_02\ID:=20,v100,z1,PKI_500\WObj:=obTROB2;
	MoveL pBack_03\ID:=30,v100,z1,PKI_500\WObj:=obTROB2;
	MoveL pBack_04\ID:=40,v100,z1,PKI_500\WObj:=obTROB2;
	MoveL pBack_05\ID:=50,v100,z1,PKI_500\WObj:=obTROB2;
	MoveL pBack_06\ID:=60,v100,z1,PKI_500\WObj:=obTROB2;
	MoveL pBack_07\ID:=70,v100,fine,PKI_500\WObj:=obTROB2;
	SyncMoveOff identBack2;
ENDPROC
ENDMODULE

--- Backups/Flexloader/RAPID/TASK3/PROGMOD/Module1.mod ---
%%%
   VERSION: 1
   LANGUAGE: ENGLISH
%%%

MODULE Module1
	VAR syncident ident1;
	PERS tasks task1{4}:=[["T_ROB1"],["T_ROB2"],["T_ROB3"],["T_ROB4"]];
	VAR syncident ident2;
	VAR syncident ident3;
	VAR syncident ident4;
	VAR syncident ident5;
	VAR syncident ident6;
	PERS tasks task4{3}:=[["T_ROB1"],["T_ROB2"],["T_ROB3"]];
	VAR syncident ident7;
	VAR syncident ident8;
	VAR syncident ident9;
	CONST robtarget pUnder_01:=[[12.828924685,255.080811168,148.825394481],[0.01722941,-0.966492314,0.004340897,-0.256079893],[0,-1,0,0],[9E+09,9E+09,9E+09,9E+09,9E+09,9E+09]];
	PERS tooldata PKI_500:=[TRUE,[[126.925343398,0,389.787472308],[0.898794046,0,0.438371147,0]],[1,[0,0,0.1],[1,0,0,0],0,0,0]];
	PERS wobjdata obTROB3:=[FALSE,FALSE,"ROB_1",[[0,0,0],[1,0,0,0]],[[0,0,0],[1,0,0,0]]];
	VAR syncident identUnder1;
	PERS tasks task2{2}:=[["T_ROB2"],["T_ROB3"]];
	CONST robtarget pUnder_02:=[[62.343632748,258.188940716,62],[0.017229379,-0.966492374,0.004340901,-0.256079667],[0,-1,0,0],[9E+09,9E+09,9E+09,9E+09,9E+09,9E+09]];
	CONST robtarget pUnder_03:=[[57.640260933,231.434848221,62],[0.017229379,-0.966492374,0.004340901,-0.256079667],[0,-1,0,0],[9E+09,9E+09,9E+09,9E+09,9E+09,9E+09]];
	CONST robtarget pUnder_04:=[[52.975980915,204.903120784,62],[0.017229379,-0.966492374,0.004340901,-0.256079667],[0,-1,0,0],[9E+09,9E+09,9E+09,9E+09,9E+09,9E+09]];
	CONST robtarget pUnder_05:=[[48.058420511,176.930663776,62],[0.017229379,-0.966492374,0.004340901,-0.256079667],[0,-1,0,0],[9E+09,9E+09,9E+09,9E+09,9E+09,9E+09]];
	CONST robtarget pUnder_06:=[[42.296035648,144.15260929,62],[0.017229379,-0.966492374,0.004340901,-0.256079667],[0,-1,0,0],[9E+09,9E+09,9E+09,9E+09,9E+09,9E+09]];
	CONST robtarget pUnder_07:=[[37.054432322,114.33690564,62],[0.017229379,-0.966492374,0.004340901,-0.256079667],[0,-1,0,0],[9E+09,9E+09,9E+09,9E+09,9E+09,9E+09]];
	CONST robtarget pUnder_08:=[[-12.460318135,111.228828412,148.825249436],[0.0172293,-0.966492333,0.004340891,-0.256079826],[0,-1,0,0],[9E+09,9E+09,9E+09,9E+09,9E+09,9E+09]];
	VAR syncident identUnder2;
	CONST robtarget pHome:=[[2488.332629759,582.160430805,1683.763976913],[0.004349692,-0.952816716,-0.133910927,0.272377036],[0,0,-1,0],[9E+09,9E+09,9E+09,9E+09,9E+09,9E+09]];
	CONST robtarget pTop_01:=[[-1.28070745,491.488881963,-0.699877698],[0.243210749,-0.588360583,-0.267180944,-0.723391111],[0,-1,0,0],[9E+09,9E+09,9E+09,9E+09,9E+09,9E+09]];
	CONST robtarget pTop_02:=[[42,525,8.932966855],[0.243210749,-0.588360583,-0.267180944,-0.723391111],[0,-1,0,0],[9E+09,9E+09,9E+09,9E+09,9E+09,9E+09]];
	VAR syncident identTop1;
	PERS tasks task3{3}:=[["T_ROB2"],["T_ROB3"],["T_ROB4"]];
	CONST robtarget pTop_03:=[[42,525,22.263152842],[0.243210749,-0.588360583,-0.267180944,-0.723391111],[0,-1,0,0],[9E+09,9E+09,9E+09,9E+09,9E+09,9E+09]];
	CONST robtarget pTop_04:=[[42,525,34.514047066],[0.243210749,-0.588360583,-0.267180944,-0.723391111],[0,-1,0,0],[9E+09,9E+09,9E+09,9E+09,9E+09,9E+09]];
	CONST robtarget pTop_05:=[[42,525,48.731913202],[0.243210749,-0.588360583,-0.267180944,-0.723391111],[0,-1,0,0],[9E+09,9E+09,9E+09,9E+09,9E+09,9E+09]];
	CONST robtarget pTop_06:=[[42,525,66.013657399],[0.243210749,-0.588360583,-0.267180944,-0.723391111],[0,-1,0,0],[9E+09,9E+09,9E+09,9E+09,9E+09,9E+09]];
	VAR syncident identTop2;
	CONST robtarget pTop_07:=[[-43.426413308,480.709402212,47.835243122],[0.243210749,-0.588360583,-0.267180944,-0.723391111],[0,-1,0,0],[9E+09,9E+09,9E+09,9E+09,9E+09,9E+09]];
	CONST robtarget pCurve_01:=[[-14.673994295,711.490040902,-16.893581967],[0.388515263,0.651173395,-0.054505115,0.649660136],[-1,-2,1,1],[9E+09,9E+09,9E+09,9E+09,9E+09,9E+09]];
	VAR syncident identCurve1;
	CONST robtarget pCurve_02:=[[64.969440267,648.464007435,-3.930130656],[0.388515305,0.651173375,-0.054505111,0.649660131],[-1,-2,1,1],[9E+09,9E+09,9E+09,9E+09,9E+09,9E+09]];
	CONST robtarget pCurve_03:=[[64.668891972,648.328807123,21.067711104],[0.3885153,0.651173377,-0.054505115,0.649660132],[-1,-2,1,1],[9E+09,9E+09,9E+09,9E+09,9E+09,9E+09]];
	CONST robtarget pCurve_04:=[[64.346339919,641.26950439,52.859645606],[0.382183452,0.754021312,0.110905328,0.522577917],[-1,-1,0,1],[9E+09,9E+09,9E+09,9E+09,9E+09,9E+09]];
	CONST robtarget pCurve_05:=[[64.202345399,621.698943338,78.891145179],[0.345890713,0.796812791,0.116503065,0.481535074],[-1,-1,0,1],[9E+09,9E+09,9E+09,9E+09,9E+09,9E+09]];
	CONST robtarget pCurve_06:=[[64.262300991,593.118173134,94.505264445],[0.345890712,0.796812802,0.116503136,0.481535039],[-1,-1,0,1],[9E+09,9E+09,9E+09,9E+09,9E+09,9E+09]];
	CONST robtarget pCurve_07:=[[64.417293699,570.916306572,97.652560093],[0.34589071,0.796812791,0.116503029,0.481535083],[-1,-1,0,1],[9E+09,9E+09,9E+09,9E+09,9E+09,9E+09]];
	CONST robtarget pCurve_08:=[[65.680062895,427.194143701,96.563249942],[0.345890732,0.796812791,0.116503045,0.481535064],[-1,-1,0,1],[9E+09,9E+09,9E+09,9E+09,9E+09,9E+09]];
	CONST robtarget pCurve_09:=[[65.871340139,411.735801615,91.846676042],[0.345890718,0.796812789,0.116503105,0.481535063],[-1,-1,0,1],[9E+09,9E+09,9E+09,9E+09,9E+09,9E+09]];
	CONST robtarget pCurve_10:=[[66.71351509,354.083378669,63.607302433],[0.345890742,0.796812788,0.116503099,0.481535049],[-1,-1,0,1],[9E+09,9E+09,9E+09,9E+09,9E+09,9E+09]];
	CONST robtarget pCurve_11:=[[66.868323931,339.314344733,61.426228634],[0.345890713,0.796812783,0.116503125,0.481535072],[-1,-1,0,1],[9E+09,9E+09,9E+09,9E+09,9E+09,9E+09]];
	CONST robtarget pCurve_12:=[[67.305924592,289.342524786,61.161160892],[0.345890727,0.796812773,0.116503069,0.481535091],[0,-1,0,1],[9E+09,9E+09,9E+09,9E+09,9E+09,9E+09]];
	VAR syncident identCurve2;
	CONST robtarget pCurve_13:=[[-31.990757531,282.227077423,145.683581488],[0.345890469,0.796812896,0.116503052,0.481535078],[0,-1,0,1],[9E+09,9E+09,9E+09,9E+09,9E+09,9E+09]];
	CONST robtarget pEdge_01:=[[-81.214404833,187.938555965,111.040053018],[0.025535838,-0.989726688,0.004582217,-0.140598745],[0,-1,0,0],[9E+09,9E+09,9E+09,9E+09,9E+09,9E+09]];
	VAR syncident identEdge1;
	CONST robtarget pEdge_02:=[[-29.612709305,190.943115239,61.621398746],[0.025535856,-0.98972668,0.004582227,-0.140598798],[0,-1,0,0],[9E+09,9E+09,9E+09,9E+09,9E+09,9E+09]];
	CONST robtarget pEdge_03:=[[-24.246494743,221.478899314,61.621785494],[0.025535876,-0.989726681,0.004582217,-0.140598785],[0,-1,0,0],[9E+09,9E+09,9E+09,9E+09,9E+09,9E+09]];
	CONST robtarget pEdge_04:=[[-18.989468125,251.393590194,61.622006852],[0.025535846,-0.989726682,0.00458224,-0.140598787],[0,-1,0,0],[9E+09,9E+09,9E+09,9E+09,9E+09,9E+09]];
	CONST robtarget pEdge_05:=[[-14.886702199,280.123923045,61.622566289],[0.025535865,-0.989726682,0.004582212,-0.140598783],[0,-1,0,0],[9E+09,9E+09,9E+09,9E+09,9E+09,9E+09]];
	CONST robtarget pEdge_06:=[[-14.888544799,308.636563639,61.622904345],[0.025535846,-0.989726683,0.00458221,-0.140598783],[0,-1,0,0],[9E+09,9E+09,9E+09,9E+09,9E+09,9E+09]];
	CONST robtarget pEdge_07:=[[-14.890348444,336.243269246,61.623380731],[0.025535841,-0.98972668,0.004582211,-0.1405988],[0,-1,0,0],[9E+09,9E+09,9E+09,9E+09,9E+09,9E+09]];
	CONST robtarget pEdge_08:=[[0.949022929,362.848749824,67.672524711],[0.025535842,-0.989726682,0.004582233,-0.140598785],[0,-1,0,0],[9E+09,9E+09,9E+09,9E+09,9E+09,9E+09]];
	CONST robtarget pEdge_09:=[[13.562331685,385.270609482,78.88309434],[0.025535836,-0.989726679,0.004582225,-0.140598806],[0,-1,0,0],[9E+09,9E+09,9E+09,9E+09,9E+09,9E+09]];
	CONST robtarget pEdge_10:=[[26.617617739,408.477924597,90.486502096],[0.025535828,-0.989726681,0.004582225,-0.140598796],[0,-1,0,0],[9E+09,9E+09,9E+09,9E+09,9E+09,9E+09]];
	CONST robtarget pEdge_11:=[[38.104972767,431.049736999,96.530678551],[0.025535841,-0.989726681,0.004582219,-0.140598796],[0,-1,0,0],[9E+09,9E+09,9E+09,9E+09,9E+09,9E+09]];
	CONST robtarget pEdge_12:=[[47.057621533,451.802110715,96.476177857],[0.025535798,-0.989726681,0.004582237,-0.140598799],[0,-1,0,0],[9E+09,9E+09,9E+09,9E+09,9E+09,9E+09]];
	CONST robtarget pEdge_13:=[[47.057249782,478.930519197,96.279515539],[0.025535856,-0.98972668,0.004582212,-0.140598796],[0,-1,0,0],[9E+09,9E+09,9E+09,9E+09,9E+09,9E+09]];
	CONST robtarget pEdge_14:=[[47.062521824,502.357435584,95.41142351],[0.025535831,-0.989726681,0.004582227,-0.140598798],[0,-1,0,0],[9E+09,9E+09,9E+09,9E+09,9E+09,9E+09]];
	CONST robtarget pEdge_15:=[[47.050756662,524.805557825,96.763928441],[0.025535834,-0.98972668,0.004582219,-0.140598799],[0,-1,0,0],[9E+09,9E+09,9E+09,9E+09,9E+09,9E+09]];
	VAR syncident identEdge2;
	CONST robtarget pEdge_16:=[[0.091457448,522.071327251,141.736609031],[0.025535838,-0.989726688,0.004582217,-0.140598745],[0,-1,0,0],[9E+09,9E+09,9E+09,9E+09,9E+09,9E+09]];
	VAR syncident identRing1;
	CONST robtarget pRing_01:=[[19.413763571,525.046564251,-107.310976223],[0.112125285,0.707925782,0.05737525,0.69496553],[0,0,-1,0],[9E+09,9E+09,9E+09,9E+09,9E+09,9E+09]];
	CONST robtarget pRing_02:=[[19.41228442,547.181655042,-108.027190051],[0.112125282,0.707925793,0.057375248,0.69496552],[0,0,-1,0],[9E+09,9E+09,9E+09,9E+09,9E+09,9E+09]];
	CONST robtarget pRing_03:=[[19.411017486,572.342907748,-94.631031476],[0.112125279,0.707925794,0.05737526,0.694965518],[-1,0,-1,0],[9E+09,9E+09,9E+09,9E+09,9E+09,9E+09]];
	CONST robtarget pRing_04:=[[19.409619957,595.082981555,-92.404501187],[0.112125289,0.707925799,0.057375223,0.694965514],[-1,0,-1,0],[9E+09,9E+09,9E+09,9E+09,9E+09,9E+09]];
	CONST robtarget pRing_05:=[[19.408023795,617.982695312,-98.41566303],[0.112125292,0.707925787,0.057375226,0.694965526],[-1,0,-1,0],[9E+09,9E+09,9E+09,9E+09,9E+09,9E+09]];
	CONST robtarget pRing_06:=[[19.40684196,632.882471871,-108.000978329],[0.112125291,0.707925781,0.057375249,0.69496553],[-1,0,-1,0],[9E+09,9E+09,9E+09,9E+09,9E+09,9E+09]];
	CONST robtarget pRing_07:=[[19.405893663,647.046556804,-107.5837926],[0.11212529,0.70792579,0.05737524,0.694965523],[-1,0,-1,0],[9E+09,9E+09,9E+09,9E+09,9E+09,9E+09]];
	VAR syncident identRing2;
	VAR syncident identBack1;
	CONST robtarget pBack_01:=[[41.352399675,-523.402928259,-106.952495913],[0.694900022,0.05761516,-0.707879949,-0.112696186],[0,0,-1,0],[9E+09,9E+09,9E+09,9E+09,9E+09,9E+09]];
	CONST robtarget pBack_02:=[[42.025569431,-545.962705591,-108.231256867],[0.694900029,0.057615167,-0.707879942,-0.112696185],[0,0,-1,0],[9E+09,9E+09,9E+09,9E+09,9E+09,9E+09]];
	CONST robtarget pBack_03:=[[42.026789538,-560.963026834,-98.938676351],[0.694900034,0.057615154,-0.707879937,-0.112696192],[0,0,-1,0],[9E+09,9E+09,9E+09,9E+09,9E+09,9E+09]];
	CONST robtarget pBack_04:=[[42.028360501,-576.697278525,-93.586103273],[0.694900029,0.057615142,-0.707879943,-0.11269619],[-1,0,-1,0],[9E+09,9E+09,9E+09,9E+09,9E+09,9E+09]];
	CONST robtarget pBack_05:=[[42.031087654,-605.790329385,-94.1859927],[0.694900037,0.057615154,-0.707879933,-0.112696198],[-1,0,-1,0],[9E+09,9E+09,9E+09,9E+09,9E+09,9E+09]];
	CONST robtarget pBack_06:=[[42.058608843,-631.783217498,-107.31836637],[0.694900023,0.057615154,-0.707879949,-0.112696182],[-1,0,-1,0],[9E+09,9E+09,9E+09,9E+09,9E+09,9E+09]];
	CONST robtarget pBack_07:=[[41.373495193,-652.531679802,-108.338921383],[0.694900021,0.057615166,-0.70787995,-0.11269618],[-1,0,-1,0],[9E+09,9E+09,9E+09,9E+09,9E+09,9E+09]];
	VAR syncident identBack2;

PROC main()
	WaitSyncTask ident1,task1;
	FromHome;
	PartTop;
	PartCurve;
	ToHome;
	WaitSyncTask ident2,task1;
	WaitSyncTask ident3,task1;
	FromHome;
	PartUnder;
	WaitSyncTask ident4,task1;
	PartEdge;
	ToHome;
	WaitSyncTask ident5,task1;
	WaitSyncTask ident6,task1;
	FromHome;
	PartRing;
	ToHome;
	WaitSyncTask ident7,task1;
	WaitSyncTask ident8,task1;
	FromHome;
	PartBack;
	ToHome;
	WaitSyncTask ident9,task1;
ENDPROC

PROC PartUnder()
	MoveJ pUnder_01,vmax,fine,PKI_500\WObj:=obTROB3;
	SyncMoveOn identUnder1,task2;
	MoveL pUnder_02\ID:=10,v500,z100,PKI_500\WObj:=obTROB3;
	MoveL pUnder_03\ID:=20,v500,z100,PKI_500\WObj:=obTROB3;
	MoveL pUnder_04\ID:=30,v500,z100,PKI_500\WObj:=obTROB3;
	MoveL pUnder_05\ID:=40,v500,z100,PKI_500\WObj:=obTROB3;
	MoveL pUnder_06\ID:=50,v500,z100,PKI_500\WObj:=obTROB3;
	MoveL pUnder_07\ID:=60,v500,z100,PKI_500\WObj:=obTROB3;
	MoveL pUnder_08\ID:=70,v500,fine,PKI_500\WObj:=obTROB3;
	SyncMoveOff identUnder2;
ENDPROC

PROC FromHome()
	MoveJ pHome,vmax,fine,PKI_500\WObj:=wobj0;
ENDPROC

PROC ToHome()
	MoveJ pHome,vmax,fine,PKI_500\WObj:=wobj0;
ENDPROC

PROC PartTop()
	MoveJ pTop_01,vmax,z100,PKI_500\WObj:=obTROB3;
	MoveL pTop_02,v500,fine,PKI_500\WObj:=obTROB3;
	SyncMoveOn identTop1,task3;
	MoveL pTop_03\ID:=10,v500,z1,PKI_500\WObj:=obTROB3;
	MoveL pTop_04\ID:=20,v500,z1,PKI_500\WObj:=obTROB3;
	MoveL pTop_05\ID:=30,v500,z1,PKI_500\WObj:=obTROB3;
	MoveL pTop_06\ID:=40,v500,fine,PKI_500\WObj:=obTROB3;
	SyncMoveOff identTop2;
	MoveL pTop_07,v500,z100,PKI_500\WObj:=obTROB3;
ENDPROC

PROC PartCurve()
	MoveJ pCurve_01,v1000,z100,PKI_500\WObj:=obTROB3;
	SyncMoveOn identCurve1,task2;
	MoveL pCurve_02\ID:=20,v500,z100,PKI_500\WObj:=obTROB3;
	MoveL pCurve_03\ID:=30,v500,z100,PKI_500\WObj:=obTROB3;
	MoveL pCurve_04\ID:=40,v500,z100,PKI_500\WObj:=obTROB3;
	MoveL pCurve_05\ID:=50,v500,z100,PKI_500\WObj:=obTROB3;
	MoveL pCurve_06\ID:=60,v500,z100,PKI_500\WObj:=obTROB3;
	MoveL pCurve_07\ID:=70,v500,z100,PKI_500\WObj:=obTROB3;
	MoveL pCurve_08\ID:=80,v500,z100,PKI_500\WObj:=obTROB3;
	MoveL pCurve_09\ID:=90,v500,z100,PKI_500\WObj:=obTROB3;
	MoveL pCurve_10\ID:=100,v500,z100,PKI_500\WObj:=obTROB3;
	MoveL pCurve_11\ID:=110,v500,z100,PKI_500\WObj:=obTROB3;
	MoveL pCurve_12\ID:=120,v500,fine,PKI_500\WObj:=obTROB3;
	SyncMoveOff identCurve2;
	MoveL pCurve_13,v1000,z100,PKI_500\WObj:=obTROB3;
ENDPROC

PROC PartEdge()
	MoveJ pEdge_01,v1000,fine,PKI_500\WObj:=obTROB3;
	SyncMoveOn identEdge1,task3;
	MoveL pEdge_02\ID:=10,v1000,z100,PKI_500\WObj:=obTROB3;
	MoveL pEdge_03\ID:=20,v1000,z100,PKI_500\WObj:=obTROB3;
	MoveL pEdge_04\ID:=30,v1000,z100,PKI_500\WObj:=obTROB3;
	MoveL pEdge_05\ID:=40,v1000,z100,PKI_500\WObj:=obTROB3;
	MoveL pEdge_06\ID:=50,v1000,z100,PKI_500\WObj:=obTROB3;
	MoveL pEdge_07\ID:=60,v1000,z100,PKI_500\WObj:=obTROB3;
	MoveL pEdge_08\ID:=70,v1000,z100,PKI_500\WObj:=obTROB3;
	MoveL pEdge_09\ID:=80,v1000,z100,PKI_500\WObj:=obTROB3;
	MoveL pEdge_10\ID:=90,v1000,z100,PKI_500\WObj:=obTROB3;
	MoveL pEdge_11\ID:=100,v1000,z100,PKI_500\WObj:=obTROB3;
	MoveL pEdge_12\ID:=110,v1000,z100,PKI_500\WObj:=obTROB3;
	MoveL pEdge_13\ID:=120,v1000,z100,PKI_500\WObj:=obTROB3;
	MoveL pEdge_14\ID:=130,v1000,z100,PKI_500\WObj:=obTROB3;
	MoveL pEdge_15\ID:=140,v1000,fine,PKI_500\WObj:=obTROB3;
	SyncMoveOff identEdge2;
	MoveL pEdge_16,v1000,z100,PKI_500\WObj:=obTROB3;
ENDPROC

PROC PartRing()
	SyncMoveOn identRing1,task2;
	MoveL pRing_01\ID:=10,v1000,z100,PKI_500\WObj:=obTROB3;
	MoveL pRing_02\ID:=20,v1000,z100,PKI_500\WObj:=obTROB3;
	MoveL pRing_03\ID:=30,v1000,z100,PKI_500\WObj:=obTROB3;
	MoveL pRing_04\ID:=40,v1000,z100,PKI_500\WObj:=obTROB3;
	MoveL pRing_05\ID:=50,v1000,z100,PKI_500\WObj:=obTROB3;
	MoveL pRing_06\ID:=60,v1000,z100,PKI_500\WObj:=obTROB3;
	MoveL pRing_07\ID:=70,v1000,fine,PKI_500\WObj:=obTROB3;
	SyncMoveOff identRing2;
ENDPROC

PROC PartBack()
	SyncMoveOn identBack1,task2;
	MoveL pBack_01\ID:=10,v1000,z100,PKI_500\WObj:=obTROB3;
	MoveL pBack_02\ID:=20,v1000,z100,PKI_500\WObj:=obTROB3;
	MoveL pBack_03\ID:=30,v1000,z100,PKI_500\WObj:=obTROB3;
	MoveL pBack_04\ID:=40,v1000,z100,PKI_500\WObj:=obTROB3;
	MoveL pBack_05\ID:=50,v1000,z100,PKI_500\WObj:=obTROB3;
	MoveL pBack_06\ID:=60,v1000,z100,PKI_500\WObj:=obTROB3;
	MoveL pBack_07\ID:=70,v1000,fine,PKI_500\WObj:=obTROB3;
	SyncMoveOff identBack2;
ENDPROC
ENDMODULE

--- Backups/Flexloader/RAPID/TASK4/PROGMOD/module1.mod ---
%%%
   VERSION: 1
   LANGUAGE: ENGLISH
%%%

MODULE module1
	VAR syncident ident1;
	PERS tasks task1{4}:=[["T_ROB1"],["T_ROB2"],["T_ROB3"],["T_ROB4"]];
	VAR syncident ident2;
	VAR syncident ident3;
	VAR syncident ident4;
	VAR syncident ident5;
	VAR syncident ident6;
	VAR syncident ident7;
	VAR syncident ident8;
	VAR syncident ident9;
	CONST robtarget pHome:=[[3875.36318289,-110.332841993,1402.722430931],[0.103374944,0.741683742,-0.013589891,0.662596531],[0,0,1,5],[9E+09,9E+09,9E+09,9E+09,9E+09,9E+09]];
	PERS tooldata PKI_500:=[TRUE,[[126.925343398,0,389.787472308],[0.898794046,0,0.438371147,0]],[1,[0,0,0.1],[1,0,0,0],0,0,0]];
	CONST robtarget pTop_01:=[[-53.933322356,-50.370197982,124.897551156],[0.02321001,-0.902367702,-0.014854786,-0.430085063],[-1,0,1,0],[9E+09,9E+09,9E+09,9E+09,9E+09,9E+09]];
	PERS wobjdata obTROB4:=[FALSE,FALSE,"ROB_1",[[0,0,0],[1,0,0,0]],[[0,0,0],[1,0,0,0]]];
	VAR syncident identTop1;
	PERS tasks task3{3}:=[["T_ROB2"],["T_ROB3"],["T_ROB4"]];
	CONST robtarget pTop_02:=[[23.616622868,-44.90363802,62],[0.023209166,-0.9023677,-0.014853952,-0.430085141],[-1,0,1,0],[9E+09,9E+09,9E+09,9E+09,9E+09,9E+09]];
	CONST robtarget pTop_03:=[[9.041580609,-27.723854217,62],[0.023209166,-0.9023677,-0.014853952,-0.430085141],[0,-1,2,0],[9E+09,9E+09,9E+09,9E+09,9E+09,9E+09]];
	CONST robtarget pTop_04:=[[-0.098576243,-2.850912622,62],[0.023209166,-0.9023677,-0.014853952,-0.430085141],[0,-1,2,0],[9E+09,9E+09,9E+09,9E+09,9E+09,9E+09]];
	CONST robtarget pTop_05:=[[8.743705294,27.213906352,62],[0.023209166,-0.9023677,-0.014853952,-0.430085141],[0,-1,2,0],[9E+09,9E+09,9E+09,9E+09,9E+09,9E+09]];
	VAR syncident identTop2;
	CONST robtarget pTop_06:=[[21.936060727,43.448780978,62],[0.023209166,-0.9023677,-0.014853952,-0.430085141],[0,-1,2,0],[9E+09,9E+09,9E+09,9E+09,9E+09,9E+09]];
	CONST robtarget pTop_07:=[[-55.613953031,37.982236208,124.897545737],[0.023210001,-0.90236772,-0.014854781,-0.430085025],[0,-1,2,0],[9E+09,9E+09,9E+09,9E+09,9E+09,9E+09]];
	CONST robtarget pEdge_01:=[[-84.438659601,-190.364208004,113.529725477],[0.025718882,-0.997608496,0.001946891,-0.06412517],[-1,0,1,0],[9E+09,9E+09,9E+09,9E+09,9E+09,9E+09]];
	VAR syncident identEdge1;
	CONST robtarget pEdge_02:=[[-30.230734504,-187.207943347,61.615009386],[0.025718882,-0.997608496,0.001946891,-0.06412517],[-1,0,1,0],[9E+09,9E+09,9E+09,9E+09,9E+09,9E+09]];
	CONST robtarget pEdge_03:=[[-35.563560424,-156.884650882,61.615738857],[0.025718882,-0.997608496,0.001946891,-0.06412517],[-1,0,1,0],[9E+09,9E+09,9E+09,9E+09,9E+09,9E+09]];
	CONST robtarget pEdge_04:=[[-40.826806863,-126.958078408,61.616225447],[0.025718882,-0.997608496,0.001946891,-0.06412517],[-1,0,1,0],[9E+09,9E+09,9E+09,9E+09,9E+09,9E+09]];
	CONST robtarget pEdge_05:=[[-42.036790435,-104.912492018,61.616704851],[0.025718882,-0.997608496,0.001946891,-0.06412517],[-1,0,1,0],[9E+09,9E+09,9E+09,9E+09,9E+09,9E+09]];
	CONST robtarget pEdge_06:=[[-40.328468341,-79.803973145,61.617043515],[0.025718882,-0.997608496,0.001946891,-0.06412517],[-1,0,1,0],[9E+09,9E+09,9E+09,9E+09,9E+09,9E+09]];
	CONST robtarget pEdge_07:=[[-45.03447588,-53.044985973,61.617581691],[0.025718882,-0.997608496,0.001946891,-0.06412517],[-1,0,1,0],[9E+09,9E+09,9E+09,9E+09,9E+09,9E+09]];
	CONST robtarget pEdge_08:=[[-49.917009105,-25.282030434,61.618215742],[0.025718882,-0.997608496,0.001946891,-0.06412517],[0,-1,2,0],[9E+09,9E+09,9E+09,9E+09,9E+09,9E+09]];
	CONST robtarget pEdge_09:=[[-54.37004905,0.039008214,61.618711845],[0.025718882,-0.997608496,0.001946891,-0.06412517],[0,-1,2,0],[9E+09,9E+09,9E+09,9E+09,9E+09,9E+09]];
	CONST robtarget pEdge_10:=[[-49.311235789,28.826390298,61.619118985],[0.025718882,-0.997608496,0.001946891,-0.06412517],[0,-1,2,0],[9E+09,9E+09,9E+09,9E+09,9E+09,9E+09]];
	CONST robtarget pEdge_11:=[[-44.709803618,55.010901647,61.619318972],[0.025718882,-0.997608496,0.001946891,-0.06412517],[0,-1,2,0],[9E+09,9E+09,9E+09,9E+09,9E+09,9E+09]];
	CONST robtarget pEdge_12:=[[-40.422836273,79.40502852,61.619668467],[0.025718882,-0.997608496,0.001946891,-0.06412517],[0,-1,2,0],[9E+09,9E+09,9E+09,9E+09,9E+09,9E+09]];
	CONST robtarget pEdge_13:=[[-41.075818412,102.758496117,61.620029836],[0.025718882,-0.997608496,0.001946891,-0.06412517],[0,-1,2,0],[9E+09,9E+09,9E+09,9E+09,9E+09,9E+09]];
	CONST robtarget pEdge_14:=[[-40.191945224,130.742368303,61.620550475],[0.025718882,-0.997608496,0.001946891,-0.06412517],[0,-1,2,0],[9E+09,9E+09,9E+09,9E+09,9E+09,9E+09]];
	CONST robtarget pEdge_15:=[[-34.743769196,161.745202367,61.620877686],[0.025718882,-0.997608496,0.001946891,-0.06412517],[0,-1,2,0],[9E+09,9E+09,9E+09,9E+09,9E+09,9E+09]];
	VAR syncident identEdge2;
	CONST robtarget pEdge_16:=[[-86.863519723,158.710435962,111.535761546],[0.025718882,-0.997608496,0.001946891,-0.06412517],[0,-1,2,0],[9E+09,9E+09,9E+09,9E+09,9E+09,9E+09]];
	CONST robtarget pClean_02:=[[3918.802527966,13.910333916,1233.885215385],[0.003707074,0.781444405,-0.012443506,0.623839771],[-1,0,2,5],[9E+09,9E+09,9E+09,9E+09,9E+09,9E+09]];
	CONST robtarget pClean_03:=[[4031.309513385,13.910333916,1233.885215385],[0.003707074,0.781444405,-0.012443506,0.623839771],[-1,0,1,5],[9E+09,9E+09,9E+09,9E+09,9E+09,9E+09]];
	CONST robtarget pClean_01:=[[3981.665484952,13.910333916,1233.885215385],[0.003707074,0.781444405,-0.012443506,0.623839771],[-1,0,2,5],[9E+09,9E+09,9E+09,9E+09,9E+09,9E+09]];
	CONST robtarget pClean_04:=[[3981.665484952,13.910333916,1181.301532419],[0.003707074,0.781444405,-0.012443506,0.623839771],[-1,0,1,5],[9E+09,9E+09,9E+09,9E+09,9E+09,9E+09]];
	CONST robtarget pClean_05:=[[3981.665484952,13.910333916,1286.282919017],[0.003707074,0.781444405,-0.012443506,0.623839771],[-1,0,2,5],[9E+09,9E+09,9E+09,9E+09,9E+09,9E+09]];
	CONST robtarget pClean_06:=[[3981.665484952,58.802264128,1233.885215385],[0.003707074,0.781444405,-0.012443506,0.623839771],[-1,0,1,5],[9E+09,9E+09,9E+09,9E+09,9E+09,9E+09]];
	CONST robtarget pClean_07:=[[3981.665484952,-26.193959875,1233.885215385],[0.003707074,0.781444405,-0.012443506,0.623839771],[0,-1,2,5],[9E+09,9E+09,9E+09,9E+09,9E+09,9E+09]];

PROC main()
	WaitSyncTask ident1,task1;
	fromBullsEye;
	PartTop;
	toBullsEye;
	WaitSyncTask ident2,task1;
	WaitSyncTask ident3,task1;
	fromBullsEye;
	WaitSyncTask ident4,task1;
	PartEdge;
	toBullsEye;
	WaitSyncTask ident5,task1;
	WaitSyncTask ident6,task1;
	fromBullsEye;
	TorchCleaner;
	toBullsEye;
	WaitSyncTask ident7,task1;
	WaitSyncTask ident8,task1;
	WaitSyncTask ident9,task1;
ENDPROC

PROC toBullsEye()
	MoveJ pHome,vmax,fine,PKI_500\WObj:=wobj0;
ENDPROC

PROC fromBullsEye()
	MoveJ pHome,vmax,fine,PKI_500\WObj:=wobj0;
ENDPROC

PROC PartTop()
	MoveJ pTop_01,vmax,z10,PKI_500\WObj:=obTROB4;
	SyncMoveOn identTop1,task3;
	MoveL pTop_02\ID:=10,v500,z1,PKI_500\WObj:=obTROB4;
	MoveL pTop_03\ID:=20,v500,z1,PKI_500\WObj:=obTROB4;
	MoveL pTop_04\ID:=30,v500,z1,PKI_500\WObj:=obTROB4;
	MoveL pTop_05\ID:=40,v500,fine,PKI_500\WObj:=obTROB4;
	SyncMoveOff identTop2;
	MoveL pTop_06,v500,z10,PKI_500\WObj:=obTROB4;
	MoveL pTop_07,v500,z10,PKI_500\WObj:=obTROB4;
ENDPROC

PROC PartEdge()
	MoveJ pEdge_01,v2000,fine,PKI_500\WObj:=obTROB4;
	SyncMoveOn identEdge1,task3;
	MoveL pEdge_02\ID:=10,v1000,z100,PKI_500\WObj:=obTROB4;
	MoveL pEdge_03\ID:=20,v1000,z100,PKI_500\WObj:=obTROB4;
	MoveL pEdge_04\ID:=30,v1000,z100,PKI_500\WObj:=obTROB4;
	MoveL pEdge_05\ID:=40,v1000,z100,PKI_500\WObj:=obTROB4;
	MoveL pEdge_06\ID:=50,v1000,z100,PKI_500\WObj:=obTROB4;
	MoveL pEdge_07\ID:=60,v1000,z100,PKI_500\WObj:=obTROB4;
	MoveL pEdge_08\ID:=70,v1000,z100,PKI_500\WObj:=obTROB4;
	MoveL pEdge_09\ID:=80,v1000,z100,PKI_500\WObj:=obTROB4;
	MoveL pEdge_10\ID:=90,v1000,z100,PKI_500\WObj:=obTROB4;
	MoveL pEdge_11\ID:=100,v1000,z100,PKI_500\WObj:=obTROB4;
	MoveL pEdge_12\ID:=110,v1000,z100,PKI_500\WObj:=obTROB4;
	MoveL pEdge_13\ID:=120,v1000,z100,PKI_500\WObj:=obTROB4;
	MoveL pEdge_14\ID:=130,v1000,z100,PKI_500\WObj:=obTROB4;
	MoveL pEdge_15\ID:=140,v1000,fine,PKI_500\WObj:=obTROB4;
	SyncMoveOff identEdge2;
	MoveL pEdge_16,v1000,z100,PKI_500\WObj:=obTROB4;
ENDPROC

PROC TorchCleaner()
	MoveJ pClean_02,v1000,z100,PKI_500\WObj:=wobj0;
	MoveL pClean_03,v100,z100,PKI_500\WObj:=wobj0;
	MoveL pClean_01,v100,z100,PKI_500\WObj:=wobj0;
	MoveL pClean_04,v100,z100,PKI_500\WObj:=wobj0;
	MoveL pClean_05,v100,z100,PKI_500\WObj:=wobj0;
	MoveL pClean_01,v100,z100,PKI_500\WObj:=wobj0;
	MoveL pClean_06,v100,z100,PKI_500\WObj:=wobj0;
	MoveL pClean_07,v100,z100,PKI_500\WObj:=wobj0;
	MoveL pClean_01,v100,z100,PKI_500\WObj:=wobj0;
	MoveL pClean_02,v100,z100,PKI_500\WObj:=wobj0;
ENDPROC
ENDMODULE
